FUNCTION TryConvert_LINT_TO_ULINT : BOOL
VAR_INPUT
	in : LINT;
	out : REFERENCE TO ULINT;
END_VAR

IF in < DatatypeLimits.MIN_VALUE_OF_LINT_WHICH_CAN_BE_HELD_IN_A_ULINT THEN
	RETURN;
END_IF

out := LINT_TO_ULINT(in);
TryConvert_LINT_TO_ULINT := TRUE;

END_FUNCTION

(* stored: Version 1.1.0.1, ProductVersion 3.1.4024.12
   POU TryConvert_LINT_TO_ULINT: Id {10118863-1f0b-415a-9a77-c5eba0fe59cd}, SpecialFunc None *)
